// Mitsubishi GX Works2 project: hung_creat_plc_dich_bit_ver4   PLC: FX3U/FX3UC

PROGRAM MAIN
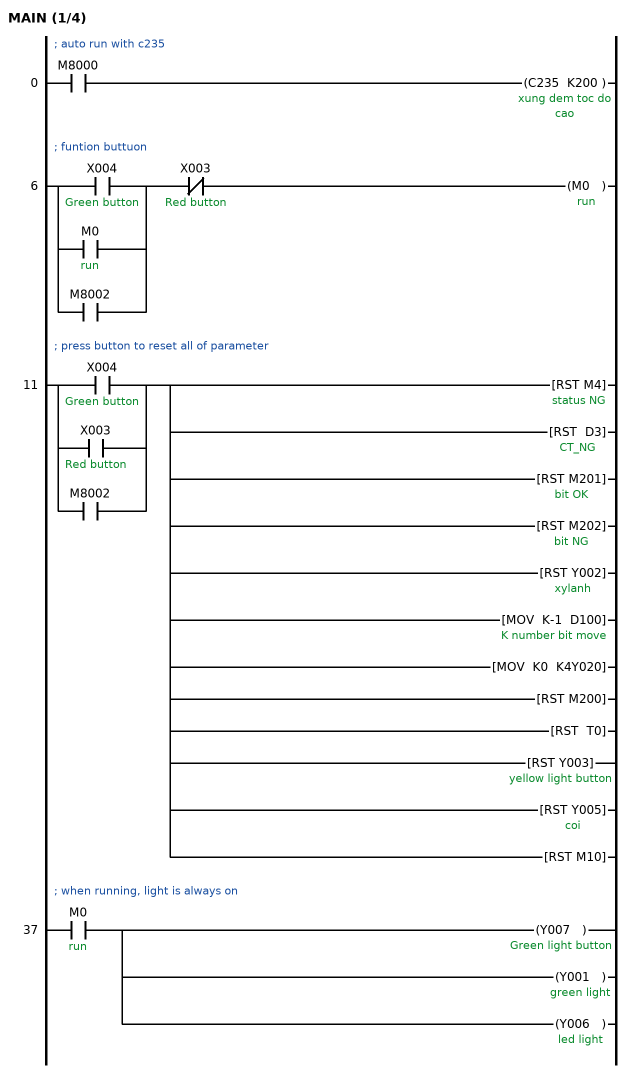
; auto run with c235
0     LD      M8000
      OUT     C235 K200  ; xung dem toc do  cao
; funtion buttuon
6     LD      X004  ; Green button
      OR      M0  ; run
      OR      M8002
      ANI     X003  ; Red button
      OUT     M0  ; run
; press button to reset all of parameter
11    LD      X004  ; Green button
      OR      X003  ; Red button
      OR      M8002
      RST     M4  ; status NG
      RST     D3  ; CT_NG
      RST     M201  ; bit OK
      RST     M202  ; bit NG
      RST     Y002  ; xylanh
      MOV     K-1 D100  ; K number bit move
      MOV     K0 K4Y020  ; move right
      RST     M200
      RST     T0
      RST     Y003  ; yellow light button
      RST     Y005  ; coi
      RST     M10
; when running, light is always on
37    LD      M0  ; run
      OUT     Y007  ; Green light button
      OUT     Y001  ; green light
      OUT     Y006  ; led light
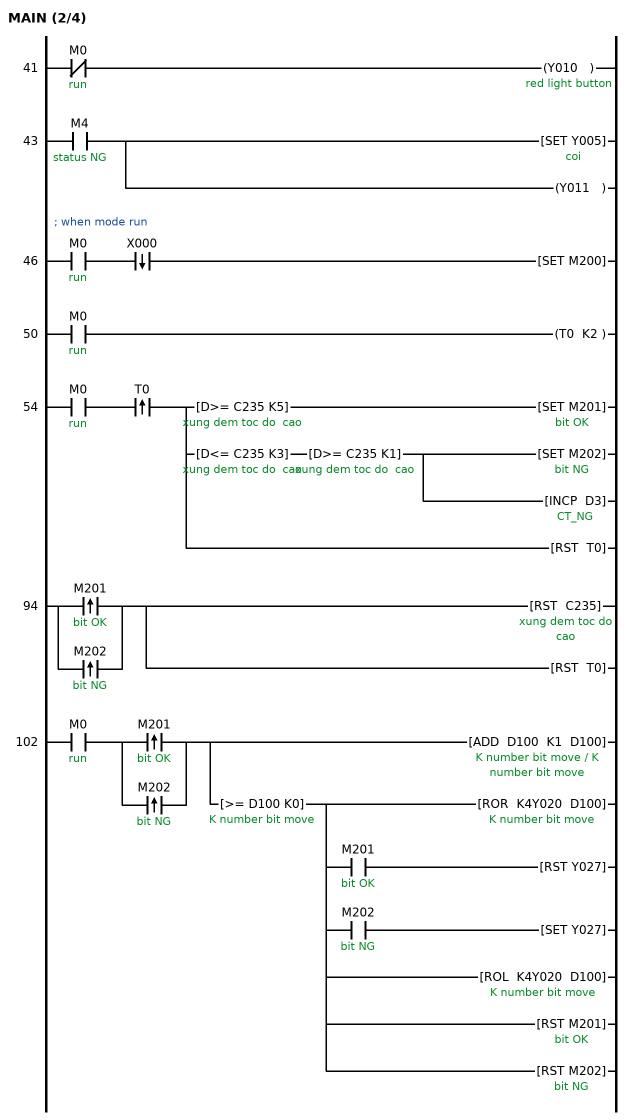
41    LDI     M0  ; run
      OUT     Y010  ; red light button
43    LD      M4  ; status NG
      SET     Y005  ; coi
      OUT     Y011
; when mode run
46    LD      M0  ; run
      ANDF    X000
      SET     M200
50    LD      M0  ; run
      OUT     T0 K2
54    LD      M0  ; run
      ANDP    T0
      MPS
      ANDD>=  C235 K5  ; xung dem toc do  cao
      SET     M201  ; bit OK
      MRD
      ANDD<=  C235 K3  ; xung dem toc do  cao
      ANDD>=  C235 K1  ; xung dem toc do  cao
      SET     M202  ; bit NG
      INCP    D3
      MPP
      RST     T0
94    LDP     M201  ; bit OK
      ORP     M202  ; bit NG
      RST     C235  ; xung dem toc do  cao
      RST     T0
102   LD      M0  ; run
      LDP     M201  ; bit OK
      ORP     M202  ; bit NG
      ANB
      ADD     D100 K1 D100
      AND>=   D100 K0  ; K number bit move
      ROR     K4Y020 D100
      MPS
      AND     M201  ; bit OK
      RST     Y027
      MRD
      AND     M202  ; bit NG
      SET     Y027
      MPP
      ROL     K4Y020 D100
      RST     M201  ; bit OK
      RST     M202  ; bit NG
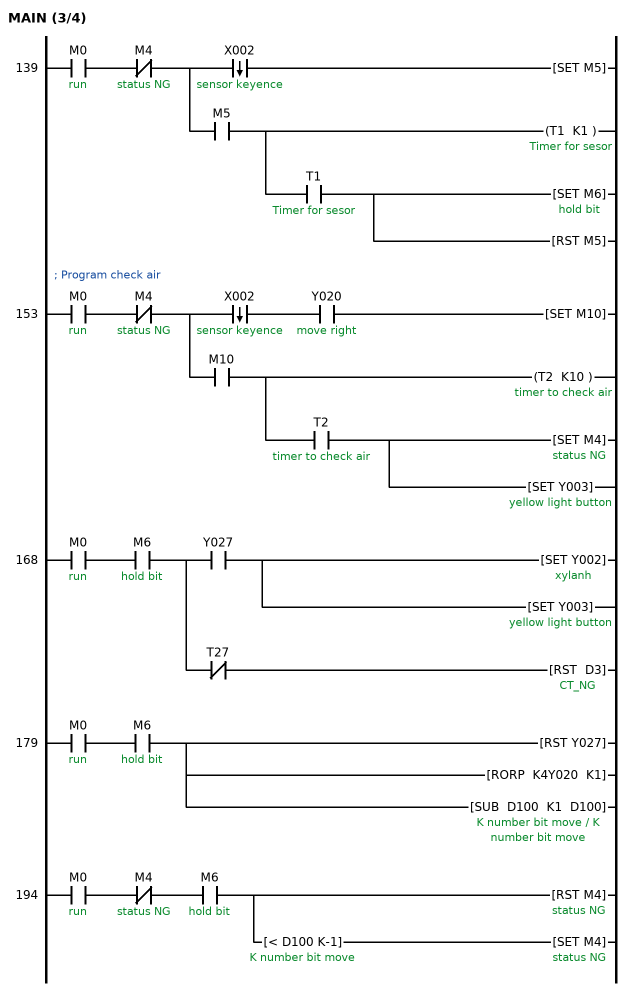
139   LD      M0  ; run
      ANI     M4  ; status NG
      MPS
      ANDF    X002  ; sensor keyence
      SET     M5
      MPP
      AND     M5
      OUT     T1 K1  ; Timer for sesor
      AND     T1  ; Timer for sesor
      SET     M6  ; hold bit
      RST     M5
; Program check air
153   LD      M0  ; run
      ANI     M4  ; status NG
      MPS
      ANDF    X002  ; sensor keyence
      AND     Y020  ; move right
      SET     M10
      MPP
      AND     M10
      OUT     T2 K10  ; timer to check air
      AND     T2  ; timer to check air
      SET     M4  ; status NG
      SET     Y003  ; yellow light button
168   LD      M0  ; run
      AND     M6  ; hold bit
      MPS
      AND     Y027
      SET     Y002  ; xylanh
      SET     Y003  ; yellow light button
      MPP
      ANI     T27
      RST     D3  ; CT_NG
179   LD      M0  ; run
      AND     M6  ; hold bit
      RST     Y027
      RORP    K4Y020 K1
      SUB     D100 K1 D100
194   LD      M0  ; run
      ANI     M4  ; status NG
      AND     M6  ; hold bit
      RST     M4  ; status NG
      AND<    D100 K-1  ; K number bit move
      SET     M4  ; status NG
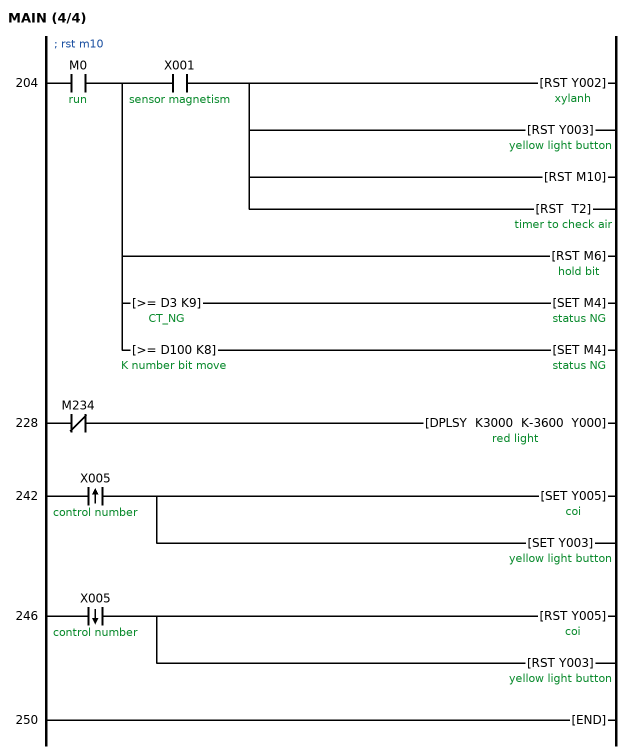
; rst m10
204   LD      M0  ; run
      MPS
      AND     X001  ; sensor magnetism
      RST     Y002  ; xylanh
      RST     Y003  ; yellow light button
      RST     M10
      RST     T2  ; timer to check air
      MPP
      RST     M6  ; hold bit
      MPS
      AND>=   D3 K9  ; CT_NG
      SET     M4  ; status NG
      MPP
      AND>=   D100 K8  ; K number bit move
      SET     M4  ; status NG
228   LDI     M234
      DPLSY   K3000 K-3600 Y000  ; red light
242   LDP     X005  ; control number
      SET     Y005  ; coi
      SET     Y003  ; yellow light button
246   LDF     X005  ; control number
      RST     Y005  ; coi
      RST     Y003  ; yellow light button
250   END
END_PROGRAM

// device comments not shown above
D0  ; CT
M3  ; bit reset NG and OK
M100  ; BIT TO MOVE
M300  ; timer for left bit
